TYPE PaletteCmd_bits_t :
STRUCT
    releaseToTargetOffset : BIT;
    direction             : BIT;
END_STRUCT
END_TYPE

(* stored: Version 1.1.0.1, ProductVersion 3.1.4024.12
   DUT PaletteCmd_bits_t: Id {9388138e-10af-41e1-aeb2-4b8ec81ee5a6} *)
